TYPE T_Ctrl_SIf_MOD_Ilk :
STRUCT
	///interlock retraction of cylinder
	bolRetract: BOOL;
	///interlock extend of cylinder
	bolExtend: BOOL;
END_STRUCT
END_TYPE

(* stored: Version 1.1.0.1, ProductVersion 3.1.0.25
   DUT T_Ctrl_SIf_MOD_Ilk: Id {ae9e7c3f-7189-4247-832f-64c2e1c25547} *)
